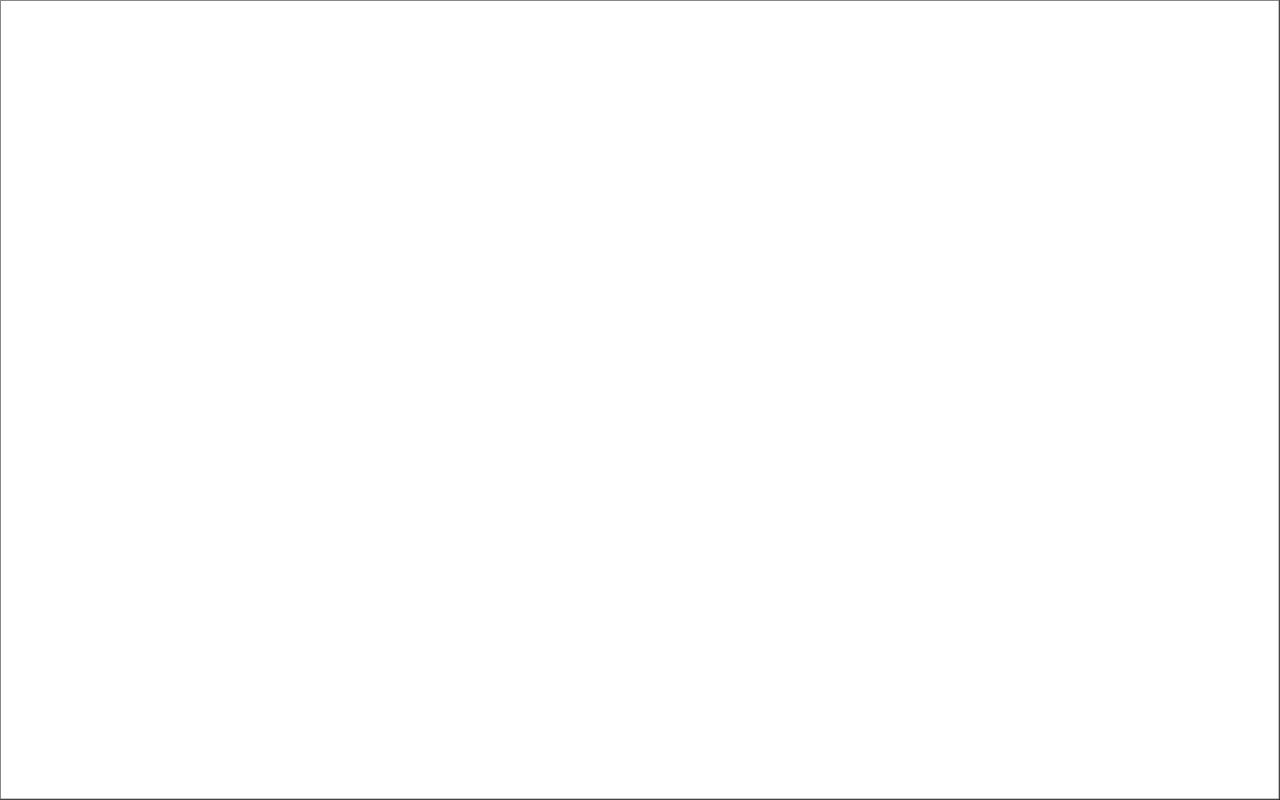
VISUALIZATION SemiAuto  // 1280x800
    Rectangle (0,0 1280x800)
END_VISUALIZATION

(* stored: Version 1.1.0.1, ProductVersion 3.1.4024.5
   Visu SemiAuto: Id {49da977c-55e0-4e44-8992-2a040fff7bb6} *)
